FUNCTION_BLOCK "turnTable90_Dual"
{ S7_Optimized_Access := 'FALSE' }
VERSION : 0.1
   VAR_INPUT
      usrBtn_Prd { ExternalVisible := 'False'} : Bool;   // User Button. Press (True) to initiate product send.
      usrBtn_DHS { ExternalVisible := 'False'} : Bool;   // Dual-hand start button input. True to rotate rollover cage.
      prdSens { ExternalVisible := 'False'} : Bool;   // Product Sensor near front. True-> Product present. (received rollers fwd)
      prdSens2 { ExternalVisible := 'False'} : Bool;   // Product Sensor near back. True-> Product present. (received rollers rev)
      prox_home { ExternalVisible := 'False'} : Bool;   // Proximity Sensor. True-> Table aligned with position 1 & 2.
      set_home : Bool;   // If true, Home pos is set to current encoder pos
      encoder_pos : DInt;   // Absolute encoder of 4096 counts for one turn of 360deg.
      eStop { ExternalVisible := 'False'} : Bool;   // Emergency stop button.
      vsdReady { ExternalVisible := 'False'} : Bool;   // Rollers VSD Online and Ready. False-> Conveyor VSD off or in Error State.
      vsdReady_TT { ExternalVisible := 'False'} : Bool;   // TurntTable VSD Online and Ready. False-> TT VSD off or in Error State.
      xManualMode : Bool;   // Manual mode request.
      comms_from_1 { ExternalVisible := 'False'} : Int;   // Communication input from previous conveyor in line. (pos 1)
      comms_from_2 { ExternalVisible := 'False'} : Int;   // Communication input from next conveyor in line. (pos 2)
      comms_from_3 { ExternalVisible := 'False'} : Int;   // Comms from conveyor @ pos 3.
      comms_from_4 { ExternalVisible := 'False'} : Int;   // Comms from conveyor @ pos 4.
      prd_in1 { ExternalVisible := 'False'} : "Product";
      prd_in2 { ExternalVisible := 'False'} : "Product";
      prd_in3 { ExternalVisible := 'False'} : "Product";
      xAutoMode { ExternalVisible := 'False'} : Bool;   // Option: True-> TT operates automatically without user and DHS.
      xOutDir : Bool;   // Option: True-> Prd is sent to pos 4. False (default)-> To 3.
      xInDir : Bool;   // Option: True-> Prd is received from 3. False (default)-> From 1.
      xEncoderTolerance : Int := 10;
   END_VAR

   VAR_OUTPUT
      rollersFwd { ExternalVisible := 'False'} : Bool;   // True-> Conveyor belt on. Product moving forward.
      rollersRev { ExternalVisible := 'False'} : Bool;   // True-> Conveyor belt on. Product moving in reverse.
      turnTableCW { ExternalVisible := 'False'} : Bool;   // True-> Turn table turning clockwise.
      turnTableACW { ExternalVisible := 'False'} : Bool;   // True-> Turn table turning anti-clockwise.
      turnTableFast { ExternalVisible := 'False'} : Bool;   // True-> Turn table turning fast speed. False-> Slow.
      statusLed { ExternalVisible := 'False'} : Bool;   // Light Indication to user.
      comms_to_1 { ExternalVisible := 'False'} : Int;   // Communication output to previous conveyor in line. (pos 1)
      comms_to_2 { ExternalVisible := 'False'} : Int;   // Communication output to next conveyor in line. (pos 2)
      comms_to_3 { ExternalVisible := 'False'} : Int;   // Comms out to conveyor @ pos 3.
      comms_to_4 { ExternalVisible := 'False'} : Int;   // Comms out to conveyor @ pos 4.
      prd_out3 { ExternalVisible := 'False'} : "Product";
      prd_out4 { ExternalVisible := 'False'} : "Product";
      alarms_out : Word;
      alarms { ExternalAccessible := 'False'; ExternalVisible := 'False'; ExternalWritable := 'False'} AT alarms_out : Array[0..15] of Bool;
   END_VAR

   VAR
      state : Int;   // Conveyor state. 0->Startup; 1->ReadyToReceive; 2->Receiving; 3->ReadyToSend; 4->Sending; 5-> Error;
      state_prev { ExternalVisible := 'False'} : Int;   // Previous conveyor state.
      intState { ExternalVisible := 'False'} : Int;   // Internal state for nested state machine.
      turnTablePos { ExternalVisible := 'False'; ExternalWritable := 'False'} : Int;   // Either 2 (home), 3 (90deg ACW), 4 (90deg CW).
      homePosCount : DInt := 16749675;
      dipTankPos_offset : Int;
      leakTestPos_offset : Int;
      prd : "Product";
      prdOutDir { ExternalVisible := 'False'} : Bool;   // Option: True-> Prd is sent to pos 4. False-> To 3. (default)
      receiveFail { ExternalVisible := 'False'} : Int;   // 0: No Fail; 1: fail rx from pos1; 2: fail rx from pos2
      sendFail { ExternalVisible := 'False'} : Int;   // 0: No Fail; 1: fail tx fwd (ps1); 2: fail tx rev (ps2)
      t_off {OriginalPartName := 'TOF'; LibVersion := '1.0'; ExternalVisible := 'False'} : TOF;
      t_on {OriginalPartName := 'TON'; LibVersion := '1.0'; ExternalVisible := 'False'} : TON;
      m_rollersFwd : Bool;   // Manual rollers motor forward request.
      m_turn_pos4 : Bool;
      m_turn_pos3 : Bool;
   END_VAR

   VAR CONSTANT
      s_startup : Int := 0;
      s_ready_to_receive : Int := 1;
      s_receiving : Int := 2;
      s_ready_to_send : Int := 3;
      s_sending : Int := 4;
      s_reset : Int := 5;
      s_turn_12 : Int := 8;
      s_turn_34 : Int := 9;
      s_manual : Int := 10;
      m_silent : Int := 0;   // Inter-conveyor message (To both) : No message
      m_req_send : Int := 100;   // Inter-conveyor message (To next) : Request to send product
      m_perm_send : Int := 101;   // Inter-conveyor message (To prev) : Permission to send product
      m_sending : Int := 102;   // Inter-conveyor message (To next) : Currently  sending product
      c_conveyor_timeout : Time := T#25S;   // Time to wait for product to arrive or leave the conveyor
   END_VAR


BEGIN
	// 180 degree turning conveyor.
	//     2    ^
	//  3 PRD 4 |
	//     1    ^
	//
	// Uses encoder and single hom proxy to determine position
	// 2018-06: Add mode to receive prd from 3, and send to 4.

	// Handle TurnTable position
	IF (#encoder_pos > (#homePosCount - #xEncoderTolerance))
	    AND (#encoder_pos < (#homePosCount + #xEncoderTolerance)) THEN
	    #turnTablePos := 2;
	ELSIF (#encoder_pos > (#homePosCount - 1024 + #dipTankPos_offset - #xEncoderTolerance))
	    AND (#encoder_pos < (#homePosCount - 1024 + #dipTankPos_offset + #xEncoderTolerance)) THEN
	    #turnTablePos := 3;
	ELSIF (#encoder_pos > (#homePosCount + 1024 + #leakTestPos_offset - #xEncoderTolerance))
	    AND (#encoder_pos < (#homePosCount + 1024 + #leakTestPos_offset + #xEncoderTolerance)) THEN
	    #turnTablePos := 4;
	ELSE
	    #turnTablePos := 0;
	END_IF;

	IF #set_home THEN
	    #homePosCount := #encoder_pos;
	END_IF;

	IF #state <> #s_reset THEN
	    // Encoder missing or offline
	    IF #encoder_pos = 0 THEN
	        #state := #s_reset;
	        // Handle EStop and VSD error and reset conveyor.
	    ELSIF (#eStop OR NOT (#vsdReady AND #vsdReady_TT)) THEN
	        #state := #s_reset;
	    END_IF;
	END_IF;

	// Conveyor state machine.
	CASE #state OF
	    0:  // Startup
	        IF #state_prev <> #state THEN
	            #state_prev := #state;
	        END_IF;

	        IF #receiveFail <> 0 THEN
	            #state := #s_ready_to_receive;
	        ELSIF #sendFail <> 0 THEN
	            IF (#prdSens OR #prdSens2) THEN
	                #state := #s_ready_to_send;
	            ELSE
	                IF #xInDir THEN
	                    #state := #s_turn_34;
	                ELSE
	                    #state := #s_turn_12;
	                END_IF;
	            END_IF;
	        ELSIF (#prdSens OR #prdSens2) THEN
	            IF ((#turnTablePos = 3) AND NOT #prdOutDir)
	                OR ((#turnTablePos = 4) AND #prdOutDir) THEN
	                #state := #s_ready_to_send;
	            ELSE
	                #state := #s_turn_34;
	            END_IF;
	        ELSE
	            // No prd detected.
	            IF #xInDir THEN
	                IF #turnTablePos = 3 THEN
	                    #state := #s_ready_to_receive;
	                ELSE
	                    #state := #s_turn_34;
	                END_IF;
	            ELSE
	                IF #turnTablePos = 2 THEN
	                    #state := #s_ready_to_receive;
	                ELSE
	                    #state := #s_turn_12;
	                END_IF;
	            END_IF;
	        END_IF;
	        ;
	    1:  // Ready to Receive
	        IF #state_prev <> #state THEN
	            #t_on(IN := false,
	                  PT := t#1s);
	            #intState := 0;
	            #state_prev := #state;
	        END_IF;

	        IF #xManualMode THEN
	            #comms_to_1 := #m_silent;
	            #comms_to_2 := #m_silent;
	            #comms_to_3 := #m_silent;
	            #state := #s_manual;
	        ELSE
	            CASE #intState OF
	                0:  // Wait for 1,2 or 3 to request to send a product.
	                    IF #turnTablePos = 2 THEN
	                        IF #xInDir THEN
	                            #state := #s_turn_34;
	                            RETURN;
	                        END_IF;
	                        IF #comms_from_1 = #m_req_send THEN
	                            #comms_to_1 := #m_perm_send;
	                            #t_on(IN := false,
	                                  PT := t#1s);
	                            #intState := 1;
	                        ELSIF #comms_from_2 = #m_req_send THEN
	                            #comms_to_2 := #m_perm_send;
	                            #t_on(IN := false,
	                                  PT := t#1s);
	                            #intState := 1;
	                        END_IF;
	                    ELSIF #turnTablePos = 3 THEN
	                        IF NOT #xInDir THEN
	                            #state := #s_turn_12;
	                            RETURN;
	                        END_IF;
	                        IF #comms_from_3 = #m_req_send THEN
	                            #comms_to_3 := #m_perm_send;
	                            #t_on(IN := false,
	                                  PT := t#1s);
	                            #intState := 1;
	                        END_IF;
	                    END_IF;
	                    ;
	                1:  // Give permission to sending conveyor.
	                    #t_on(IN := true,
	                          PT := t#1s);
	                    IF #t_on.Q THEN
	                        #comms_to_1 := #m_silent;
	                        #comms_to_2 := #m_silent;
	                        #comms_to_3 := #m_silent;
	                        #intState := 0;
	                    ELSE
	                        IF (#comms_from_1 = #m_sending AND #comms_to_1 = #m_perm_send) OR
	                            (#comms_from_2 = #m_sending AND #comms_to_2 = #m_perm_send) OR
	                            (#comms_from_3 = #m_sending AND #comms_to_3 = #m_perm_send) THEN
	                            #state := #s_receiving;
	                        END_IF;
	                    END_IF;
	                    ;
	            END_CASE;
	        END_IF;
	        ;
	    2:  // Receiving
	        IF #state_prev <> #state THEN
	            #t_on(IN := false,
	                  PT := #c_conveyor_timeout);
	            #prdOutDir := #xOutDir;
	            IF #comms_from_1 = #m_sending THEN
	                #prd := #prd_in1;
	                #rollersFwd := true;
	            ELSIF #comms_from_2 = #m_sending THEN
	                #prd := #prd_in2;
	                #rollersRev := true;
	            ELSIF #comms_from_3 = #m_sending THEN
	                #prd := #prd_in3;
	                #rollersRev := true;
	            END_IF;
	            #state_prev := #state;
	        END_IF;

	        #t_on(IN := true,
	              PT := #c_conveyor_timeout);

	        IF (#prdSens AND #comms_from_1 = #m_sending) OR
	            (#prdSens2 AND #comms_from_2 = #m_sending) OR
	            (#prdSens2 AND #comms_from_3 = #m_sending) THEN
	            #receiveFail := 0;
	            #state := #s_turn_34;
	        ELSE
	            IF #t_on.Q THEN
	                // Timeout error - Product did not arrive in time.
	                #alarms[0] := true;
	                IF #rollersFwd THEN
	                    #receiveFail := 1;
	                ELSE
	                    IF #xInDir THEN
	                        #receiveFail := 3;
	                    ELSE
	                        #receiveFail := 2;
	                    END_IF;
	                END_IF;
	                #state := #s_reset;
	            END_IF;
	        END_IF;

	        IF #state_prev <> #state THEN
	            #comms_to_1 := #m_silent;
	            #comms_to_2 := #m_silent;
	            #comms_to_3 := #m_silent;
	            #rollersFwd := false;
	            #rollersRev := false;
	        END_IF;
	        ;
	    3:  // Ready to Send
	        IF #state_prev <> #state THEN
	            #t_on(IN := false,
	                  PT := t#1s);
	            #intState := 0;
	            #state_prev := #state;
	        END_IF;

	        IF NOT (#prdSens OR #prdSens2) THEN
	            // Product mysteriously dissapeared.
	            #comms_to_3 := #m_silent;
	            #comms_to_4 := #m_silent;
	            #alarms[2] := true;
	            #state := #s_reset;
	        ELSIF #xManualMode THEN
	            #comms_to_3 := #m_silent;
	            #comms_to_4 := #m_silent;
	            #state := #s_manual;
	        ELSE
	            CASE #intState OF
	                0:  // Wait for 1 or 2 to request to send a product.
	                    IF #usrBtn_Prd OR #xAutoMode THEN
	                        IF #prdOutDir THEN
	                            #comms_to_4 := #m_req_send;
	                        ELSE
	                            #comms_to_3 := #m_req_send;
	                        END_IF;
	                        #t_on(IN := false,
	                              PT := t#1s);
	                        #intState := 1;
	                    END_IF;
	                    ;
	                1:  // Give permission to sending conveyor.
	                    #t_on(IN := true,
	                          PT := t#1s);
	                    IF #t_on.Q THEN
	                        #comms_to_3 := #m_silent;
	                        #comms_to_4 := #m_silent;
	                        #intState := 0;
	                    ELSE
	                        IF (#comms_from_3 = #m_perm_send AND #comms_to_3 = #m_req_send) THEN
	                            #state := #s_sending;
	                        ELSIF (#comms_from_4 = #m_perm_send AND #comms_to_4 = #m_req_send) THEN
	                            #state := #s_sending;
	                        END_IF;
	                    END_IF;
	                    ;
	            END_CASE;
	        END_IF;
	        ;
	    4:  // Sending
	        IF #state_prev <> #state THEN
	            #t_on(IN := false,
	                  PT := #c_conveyor_timeout);
	            #rollersFwd := true;
	            IF #prdOutDir THEN
	                #prd_out4 := #prd;
	                #comms_to_4 := #m_sending;
	            ELSE
	                #prd_out3 := #prd;
	                #comms_to_3 := #m_sending;
	            END_IF;
	            #intState := 0;
	            #state_prev := #state;
	        END_IF;

	        #t_on(IN := true,
	              PT := #c_conveyor_timeout);

	        CASE #intState OF
	            0:  // Wait for product to reach last sensor.
	                IF (#rollersFwd AND #prdSens) THEN
	                    #intState := 1;
	                END_IF;
	                ;
	            1:  // Handle product send.
	                IF NOT #prdSens THEN
	                    IF (#prdOutDir AND (#comms_from_4 <> #m_perm_send))
	                        OR (NOT #prdOutDir AND (#comms_from_3 <> #m_perm_send)) THEN
	                        #sendFail := 0;
	                        IF #xInDir THEN
	                            #state := #s_turn_34;
	                        ELSE
	                            #state := #s_turn_12;
	                        END_IF;
	                    END_IF;
	                END_IF;
	                ;
	        END_CASE;

	        IF #t_on.Q THEN
	            // Timeout error - Product did not leave in time.
	            #alarms[1] := true;
	            #sendFail := 1;
	            #state := #s_reset;
	        END_IF;

	        IF #state_prev <> #state THEN
	            #rollersFwd := false;
	            #comms_to_3 := #m_silent;
	            #comms_to_4 := #m_silent;
	        END_IF;
	        ;
	    5:  // Reset
	        IF #state_prev <> #state THEN
	            #rollersFwd := false;
	            #turnTableACW := false;
	            #turnTableCW := false;
	            #statusLed := false;
	            #comms_to_3 := 0;
	            #comms_to_2 := 0;
	            #comms_to_1 := 0;
	            #t_on(IN := false,
	                  PT := t#2s);
	            #state_prev := #state;
	        END_IF;

	        #t_on(IN := true,
	              PT := t#2s);

	        IF #t_on.Q THEN
	            #alarms_out := 0;
	        END_IF;

	        #alarms[8] := NOT #vsdReady AND NOT #eStop;
	        #alarms[9] := NOT #vsdReady_TT AND NOT #eStop;
	        #alarms[10] := #encoder_pos = 0;

	        IF #t_on.Q
	            AND NOT #eStop
	            AND #vsdReady
	            AND #vsdReady_TT
	            AND (#encoder_pos <> 0)
	        THEN
	            #alarms_out := 0;
	            #state := #s_startup;
	        END_IF;
	        ;
	    8:  // Turning table to align with 1 & 2.
	        IF #state_prev <> #state THEN
	            #t_on(IN := false,
	                  PT := #c_conveyor_timeout);
	            IF #encoder_pos > #homePosCount THEN
	                #turnTableACW := true;
	            ELSE
	                #turnTableCW := true;
	            END_IF;
	            #turnTableFast := true;
	            #state_prev := #state;
	        END_IF;

	        #t_on(IN := true,
	              PT := #c_conveyor_timeout);

	        // slow down before pos reached
	        IF #turnTableFast THEN
	            IF #turnTableACW THEN
	                IF #encoder_pos < (#homePosCount + #xEncoderTolerance + 124) THEN
	                    #turnTableFast := false;
	                END_IF;
	            ELSE
	                IF #encoder_pos > (#homePosCount - #xEncoderTolerance - 124) THEN
	                    #turnTableFast := false;
	                END_IF;
	            END_IF;
	        END_IF;

	        IF #t_on.Q THEN
	            #alarms[3] := true;
	            #state := #s_reset;
	        ELSIF #turnTablePos = 2 THEN
	            #state := #s_ready_to_receive;
	        ELSIF #xManualMode THEN
	            #state := #s_manual;
	        END_IF;

	        IF #state_prev <> #state THEN
	            #turnTableCW := false;
	            #turnTableACW := false;
	            #turnTableFast := false;
	        END_IF;
	        ;
	    9:  // Turning table to align with 3 & 4.
	        IF #state_prev <> #state THEN
	            #t_on(IN := false,
	                  PT := #c_conveyor_timeout);
	            IF (#prdSens OR #prdSens2) AND #prdOutDir THEN
	                #turnTableCW := true; // turn to 4
	            ELSE
	                #turnTableACW := true; // turn to 3
	            END_IF;
	            #turnTableFast := true;
	            #state_prev := #state;
	        END_IF;

	        #t_on(IN := true,
	              PT := #c_conveyor_timeout);

	        // slow down before pos reached
	        IF #turnTableFast THEN
	            IF #turnTableCW THEN
	                IF #encoder_pos > (#homePosCount - #xEncoderTolerance + 900) THEN
	                    #turnTableFast := false;
	                END_IF;
	            ELSE
	                IF #encoder_pos < (#homePosCount + #xEncoderTolerance - 900) THEN
	                    #turnTableFast := false;
	                END_IF;
	            END_IF;
	        END_IF;

	        IF #t_on.Q THEN
	            #alarms[4] := true;
	            #state := #s_reset;
	        ELSIF (#turnTableCW AND (#turnTablePos = 4)) THEN
	            #state := #s_ready_to_send;
	        ELSIF (#turnTableACW AND (#turnTablePos = 3)) THEN
	            IF (#prdSens OR #prdSens2) THEN
	                #state := #s_ready_to_send;
	            ELSE
	                #state := #s_ready_to_receive;
	            END_IF;
	        ELSIF #xManualMode THEN
	            #state := #s_manual;
	        END_IF;

	        IF #state_prev <> #state THEN
	            #turnTableCW := false;
	            #turnTableACW := false;
	            #turnTableFast := false;
	        END_IF;
	        ;
	    10:  // Manual Mode
	        IF #state_prev <> #state THEN
	            #m_rollersFwd := false;
	            #m_turn_pos3 := false;
	            #m_turn_pos4 := false;
	            #state_prev := #state;
	        END_IF;

	        #rollersFwd := #m_rollersFwd;
	        #turnTableCW := #m_turn_pos4 AND (#turnTablePos <> 4) AND (#encoder_pos < (#homePosCount + 1024 + #xEncoderTolerance));
	        #turnTableACW := #m_turn_pos3 AND (#turnTablePos <> 3) AND (#encoder_pos > (#homePosCount - 1024 - #xEncoderTolerance));

	        IF NOT #xManualMode THEN
	            #state := #s_reset;
	        END_IF;

	        IF #state_prev <> #state THEN
	            #rollersFwd := false;
	            #turnTableACW := false;
	            #turnTableCW := false;

	            #m_rollersFwd := false;
	            #m_turn_pos3 := false;
	            #m_turn_pos4 := false;
	        END_IF;
	        ;
	END_CASE;

	// Encoder overrun protection.
	IF (#encoder_pos > (#homePosCount + 1200)) THEN
	    #alarms[11] := true;
	    #turnTableCW := false;
	ELSIF (#homePosCount < (#homePosCount - 1200)) THEN
	    #alarms[11] := true;
	    #turnTableACW := false;
	ELSE
	    #alarms[11] := false;
	END_IF;

END_FUNCTION_BLOCK

